// TIA Portal project "Project1" (V15.1)

(* hardware
DEVICE "S7-1200 station_1"  S7-1200 Station
   slot 0: "Rack_0"  S7-1200 Rack  Rack  V1.0
   slot 1: "PLC_1"  CPU 1214C DC/DC/DC  6ES7 214-1AG40-0XB0  V4.1
*)

// ===== PLC "PLC_1"  CPU 1214C DC/DC/DC =====

DATA_BLOCK "db"   // DB1
{ S7_Optimized_Access := 'TRUE' }
VERSION : 0.1
   VAR
      "time" : Time_Of_Day;
      current_time_of_day : Time_Of_Day;
      current_time : DTL;
      time_in_seconds : DInt;
      current_time_in_seconds : DInt;
      flag : Bool;
      flag_in_sec : Bool;
      flag_req : Bool;
   END_VAR
BEGIN
END_DATA_BLOCK

DATA_BLOCK "DB_report_time"   // DB9
{ S7_Optimized_Access := 'TRUE' }
VERSION : 0.1
   VAR
      time_array : Array[0..2] of Time_Of_Day;
      write_request : Bool;
   END_VAR
BEGIN
   time_array[0] := TOD#06:00:00;
   time_array[1] := TOD#14:00:00;
   time_array[2] := TOD#22:00:00;
END_DATA_BLOCK

FUNCTION "load" : Void   // FC1, SCL
{ S7_Optimized_Access := 'TRUE' }
VERSION : 0.1
   VAR_TEMP
      i : DInt;
   END_VAR
BEGIN

   WHILE #i < 110000 DO
       #i := #i + 1;
   END_WHILE;
END_FUNCTION

FUNCTION "tod_to_seconds" : DInt   // FC2, SCL
{ S7_Optimized_Access := 'TRUE' }
VERSION : 0.1
   VAR_INPUT
      input_time : Time_Of_Day;
   END_VAR
BEGIN

   #tod_to_seconds := TOD_TO_DINT(IN := #input_time) / 1000;
END_FUNCTION

FUNCTION "glue_volume_reporting_expiration" : Bool   // FC74, SCL
{ S7_Optimized_Access := 'TRUE' }
VERSION : 0.1
   VAR_INPUT
      time_index : Int;
      current_time : DTL;
      time_array : Array[0..2] of Time_Of_Day;
   END_VAR
   VAR CONSTANT
      trashold : Time := T#6H;
   END_VAR
BEGIN


   IF #time_index < 3
   THEN
       IF "tod_to_seconds"(DTL_TO_TOD(#current_time)) = "tod_to_seconds"(#time_array[#time_index])
       THEN
           #glue_volume_reporting_expiration := true;
       ELSE
           #glue_volume_reporting_expiration := "glue_volume_reporting_expiration"(time_index :=(#time_index + 1), current_time:=#current_time, time_array:=#time_array);
       END_IF;
   ELSE
       #glue_volume_reporting_expiration := false;
   END_IF;
END_FUNCTION

ORGANIZATION_BLOCK "Main"   // OB1, LAD, ProgramCycle
TITLE = "Main Program Sweep (Cycle)"
{ S7_Optimized_Access := 'TRUE' }
VERSION : 0.1
   VAR_INPUT
      Initial_Call : Bool;   // Initial call of this OB
      Remanence : Bool;   // =True, if remanent data are available
   END_VAR
   VAR_TEMP
      ret : Int;
      time_elapsed : Bool;
   END_VAR
BEGIN

REGION Network 1
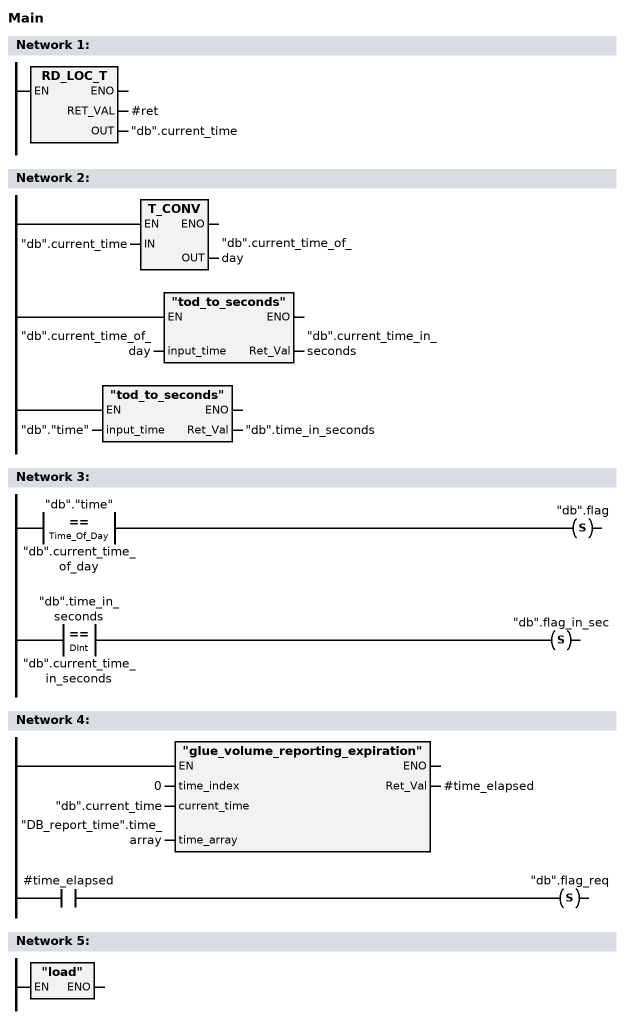
   #ret := RD_LOC_T(OUT => "db".current_time);
END_REGION

REGION Network 2
   "db".current_time_of_day := T_CONV(IN := "db".current_time);
   "db".current_time_in_seconds := "tod_to_seconds"(input_time := "db".current_time_of_day);
   "db".time_in_seconds := "tod_to_seconds"(input_time := "db"."time");
END_REGION

REGION Network 3
   RUNG wire#powerrail
      { S7_Templates := "SrcType := Time_Of_Day" } EQ_Contact(in1 := "db"."time", in2 := "db".current_time_of_day)
      S_Coil( "db".flag )
   END_RUNG
   RUNG wire#powerrail
      { S7_Templates := "SrcType := DInt" } EQ_Contact(in1 := "db".time_in_seconds, in2 := "db".current_time_in_seconds)
      S_Coil( "db".flag_in_sec )
   END_RUNG
   // the same network as SCL:
   IF "db"."time" = "db".current_time_of_day THEN "db".flag := TRUE; END_IF;
   IF "db".time_in_seconds = "db".current_time_in_seconds THEN "db".flag_in_sec := TRUE; END_IF;
END_REGION

REGION Network 4
   RUNG wire#powerrail
      "glue_volume_reporting_expiration"(time_index := 0, current_time := "db".current_time, time_array := "DB_report_time".time_array, Ret_Val => #time_elapsed)
   END_RUNG
   RUNG wire#powerrail
      Contact( #time_elapsed )
      S_Coil( "db".flag_req )
   END_RUNG
   // the same network as SCL:
   #time_elapsed := "glue_volume_reporting_expiration"(time_index := 0,
                           current_time := "db".current_time,
                           time_array := "DB_report_time".time_array);
   IF #time_elapsed THEN "db".flag_req := TRUE; END_IF;
END_REGION

REGION Network 5
   RUNG wire#powerrail
      "load"()
   END_RUNG
   // the same network as SCL:
   "load"();
END_REGION
END_ORGANIZATION_BLOCK